FUNCTION_BLOCK ThreeConCtl (* Composite Function Block Type *)
  (* Standard: 61499-2 *)
  (* Version 0.2, 2003-12-05, JHC, Rockwell Automation, Renamed from NEWCOMPFB. *)
  (* Version 0.1, 2002-01-08, JHC, Rockwell Automation, Added DLY FB as example. *)
  (* Version 0.0, 2000-05-27, JHC, Rockwell Automation *)
  (* Compiler header: package fb.rt.cs725; *)
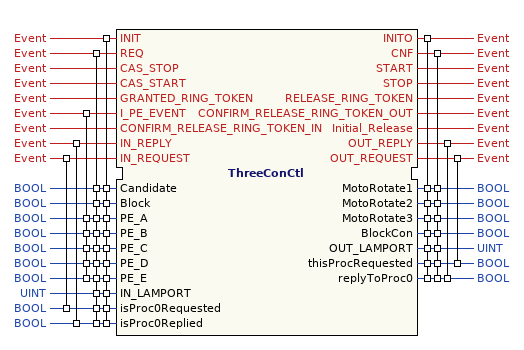
  EVENT_INPUT
    INIT WITH Candidate, Block, PE_A, PE_B, PE_C, PE_D, PE_E, isProc0Requested, IN_LAMPORT, isProc0Replied; (* Initialization Request *)
    REQ WITH Block, Candidate, PE_A, PE_B, PE_C, PE_D, PE_E, IN_LAMPORT, isProc0Requested, isProc0Replied; (* Normal Execution Request *)
    CAS_STOP;
    CAS_START;
    GRANTED_RING_TOKEN;
    I_PE_EVENT WITH PE_A, PE_B, PE_C, PE_D, PE_E;
    CONFIRM_RELEASE_RING_TOKEN_IN;
    IN_REPLY WITH isProc0Replied;
    IN_REQUEST WITH isProc0Requested;
  END_EVENT
  EVENT_OUTPUT
    INITO WITH MotoRotate1, MotoRotate2, MotoRotate3, BlockCon, thisProcRequested, replyToProc0, OUT_LAMPORT; (* Initialization Confirm *)
    CNF WITH MotoRotate1, MotoRotate2, MotoRotate3, BlockCon, OUT_LAMPORT, thisProcRequested, replyToProc0; (* Execution Confirmation *)
    START;
    STOP;
    RELEASE_RING_TOKEN;
    CONFIRM_RELEASE_RING_TOKEN_OUT;
    Initial_Release;
    OUT_REPLY WITH replyToProc0;
    OUT_REQUEST WITH thisProcRequested;
  END_EVENT
  VAR_INPUT
    Candidate : BOOL;
    Block : BOOL;
    PE_A : BOOL;
    PE_B : BOOL;
    PE_C : BOOL;
    PE_D : BOOL;
    PE_E : BOOL;
    IN_LAMPORT : UINT;
    isProc0Requested : BOOL;
    isProc0Replied : BOOL;
  END_VAR
  VAR_OUTPUT
    MotoRotate1 : BOOL;
    MotoRotate2 : BOOL;
    MotoRotate3 : BOOL;
    BlockCon : BOOL;
    OUT_LAMPORT : UINT;
    thisProcRequested : BOOL;
    replyToProc0 : BOOL;
  END_VAR
  FBS
    Conv7Ctl : ConveyorRingTokenCTL(HAS_INITIAL_TOKEN := 0);
    Conv8Ctl : ConveyorCTLMulticast(Block := 0, Candidate := 0);
    FC13 : ConveyorCTL(Block := 0, Candidate := 0);
  END_FBS
  EVENT_CONNECTIONS
    INIT TO Conv7Ctl.INIT;
    REQ TO Conv7Ctl.REQ;
    Conv7Ctl.INITO TO Conv8Ctl.INIT;
    Conv8Ctl.INITO TO FC13.INIT;
    FC13.INITO TO INITO;
    FC13.CNF TO CNF;
    REQ TO Conv8Ctl.REQ;
    REQ TO FC13.REQ;
    Conv7Ctl.CNF TO CNF;
    Conv8Ctl.CNF TO CNF;
    CAS_STOP TO Conv7Ctl.CAS_STOP;
    CAS_START TO Conv7Ctl.CAS_START;
    FC13.STOP TO STOP;
    FC13.START TO START;
    I_PE_EVENT TO Conv7Ctl.I_PE_EVENT;
    GRANTED_RING_TOKEN TO Conv7Ctl.GRANTED_RING_TOKEN;
    Conv7Ctl.RELEASE_RING_TOKEN TO RELEASE_RING_TOKEN;
    CAS_STOP TO Conv8Ctl.CAS_STOP;
    CAS_START TO Conv8Ctl.CAS_START;
    I_PE_EVENT TO Conv8Ctl.PE_EVENT;
    IN_REPLY TO Conv8Ctl.IN_REPLY;
    IN_REQUEST TO Conv8Ctl.IN_REQUEST;
    Conv8Ctl.OUT_REPLY TO OUT_REPLY;
    Conv8Ctl.OUT_REQUEST TO OUT_REQUEST;
  END_CONNECTIONS
  DATA_CONNECTIONS
    FC13.MotoRotate TO MotoRotate3;
    Conv8Ctl.MotoRotate TO MotoRotate2;
    Conv7Ctl.MotoRotate TO MotoRotate1;
    Block TO Conv7Ctl.Block;
    Conv7Ctl.BlockCon TO BlockCon;
    Candidate TO Conv7Ctl.Candidate;
    PE_C TO FC13.PE;
    PE_A TO Conv7Ctl.PE_IN;
    PE_B TO Conv7Ctl.PE_OUT;
    PE_D TO Conv8Ctl.PE_OUT;
    PE_C TO Conv8Ctl.PE_IN;
    isProc0Replied TO Conv8Ctl.isProc0Replied;
    Conv8Ctl.thisProcRequested TO thisProcRequested;
    Conv8Ctl.replyToProc0 TO replyToProc0;
    IN_LAMPORT TO Conv8Ctl.IN_LAMPORT;
    Conv8Ctl.OUT_LAMPORT TO OUT_LAMPORT;
    isProc0Requested TO Conv8Ctl.isProc0Requested;
  END_CONNECTIONS
END_FUNCTION_BLOCK
